{attribute 'GeneratedUsingTerminal: EPP3632-0001-0016'}
{attribute addProperty BoxType "EPP3632-0001-0016"}
{attribute addProperty Id "Sample_CountAT %I*UINT2"}
{attribute addProperty CRC "3934833369"}
{attribute addProperty Size "2"}
TYPE Sample_Count_EA88CAD9 :
STRUCT
	{attribute addProperty Name "Sample_Count"}
	Sample_Count AT %I* : UINT;
END_STRUCT
END_TYPE

(* stored: Version 1.2.0.0, ProductVersion 3.1.4024.9
   DUT Sample_Count_EA88CAD9: Id {93fb0348-cfc6-4274-ac3a-01f2b6ebceaf} *)
